(* Logix 5000 project; controller BallnPlate 5069-L306ERM rev 30.11; software revision 30.00 *)

TASK MainTask (periodic, rate 10 ms, priority 10, watchdog 500 ms) : MainProgram

MODULES
   Local : 5069-L306ERM (5069 0, rev 30.11)
       : 5069-IF8 (5069 3, rev 2.1, StandardDataDriven RPI 100 ms)
       : 5069-IB16 (5069 1, rev 2.1, StandardDataDriven RPI 5 ms)
       : 5069-OB16 (5069 2, rev 2.1, StandardDataDriven RPI 5 ms)
       : vendor 1 type 115 code 320 (5069 4, rev 2.1, StandardDataDriven RPI 80 ms)
END_MODULES

PROGRAM MainProgram   (* main routine Main *)
VAR
   ArduinoVoltage : DINT;
   DERV_01 : DERIVATIVE := (Gain := 1.0, RTSTime := 1);
   Desired_X_Location : DINT;
   Desired_Y_Location : DINT;
   Kd : REAL;
   Kdx : REAL;
   Kix : REAL;
   Kpx : REAL;
   LPF_01 : FILTER_LOW_PASS := (Order := 1, RTSTime := 1);
   LPF_02 : FILTER_LOW_PASS := (Order := 1, RTSTime := 1);
   MUL_01 : FBD_MATH;
   SCL_01 : SCALE;
   SCL_02 : SCALE;
   SUB_01 : FBD_MATH;
   SUB_02 : FBD_MATH;
   X_in : ALIAS FOR Local:3:I.Ch02.Data;
   Xout : ALIAS FOR Local:4:O.Ch02.Data;
   Y_in : ALIAS FOR Local:3:I.Ch00.Data;
   Yout : ALIAS FOR Local:4:O.Ch00.Data;
END_VAR

ROUTINE Main   (* function block diagram *)
   SHEET 1
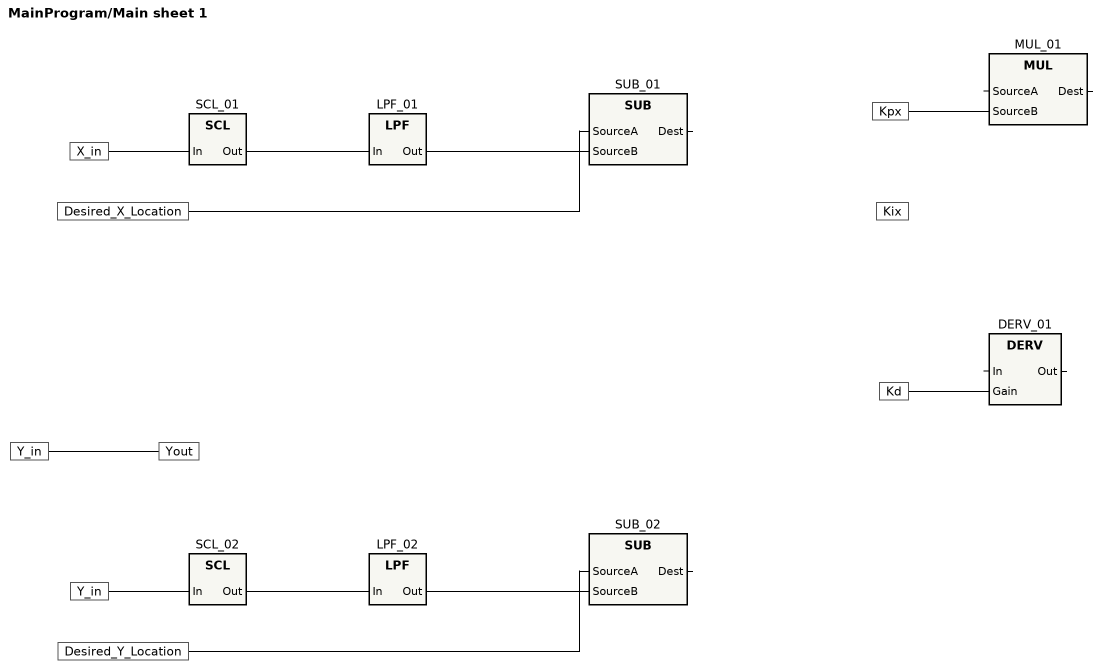
   Yout := Y_in;
   SCL_01 : SCL(In := X_in);
   SCL_02 : SCL(In := Y_in);
   LPF_01 : LPF(In := SCL_01.Out);
   LPF_02 : LPF(In := SCL_02.Out);
   SUB_01 : SUB(SourceA := Desired_X_Location, SourceB := LPF_01.Out);   // unwired pins: Dest
   SUB_02 : SUB(SourceA := Desired_Y_Location, SourceB := LPF_02.Out);   // unwired pins: Dest
   // unwired input reference Kix
   MUL_01 : MUL(SourceB := Kpx);   // unwired pins: SourceA Dest
   DERV_01 : DERV(Gain := Kd);   // unwired pins: In Out
END_ROUTINE
END_PROGRAM
